Staubli VAL3: MsgType.pjx

--- MsgType.pjx ---
Parameters version=s7.8.1 stackSize=5000 millimeterUnit=true
Program file=start.pgx
Program file=stop.pgx
Data file=MsgType.dtx

--- MsgType.dtx ---
public num PING
public num GET_VERSION
public num JOINT_POSITION
public num JOINT_TRAJ
public num JOINT_TRAJ_PT
public num JOINT_TRAJ_PT_F
public num JOINT_FEEDBACK
public num STATUS
